(* PLC project Unnamed, Unknown Unnamed 1 *)
(* stored: creationDateTime 2025-11-14T09:55:49, modificationDateTime 2026-02-01T23:59:25 *)

PROGRAM program0
  VAR
    TP0 : TP;  (* Pulse Timer *)
  END_VAR
  VAR
    InletValve1 AT %QX0.1 : BOOL;  (* Output *)
    InletValve2 AT %QX0.2 : BOOL;  (* Output *)
    Start AT %IX0.1 : BOOL;  (* Input *)
    Stop AT %IX0.2 : BOOL;  (* Input *)
    CycleOn AT %IX0.3 : BOOL;  (* Input *)
    LevelSensor1 AT %IX0.4 : BOOL;  (* Input *)
    LevelSensor2 AT %IX0.5 : BOOL;  (* Input *)
    AgitatorMotor AT %QX0.3 : BOOL;  (* Output *)
    LowLevelSensor AT %IX0.6 : BOOL;  (* Input *)
    OutletValve AT %QX0.4 : BOOL;  (* Output *)
    TemperatureSensor AT %IW0 : INT := 28;  (* Input *)
  END_VAR
  VAR
    Flag : BOOL;
  END_VAR
  VAR
    Heater AT %QX1.0 : BOOL;  (* Output *)
  END_VAR

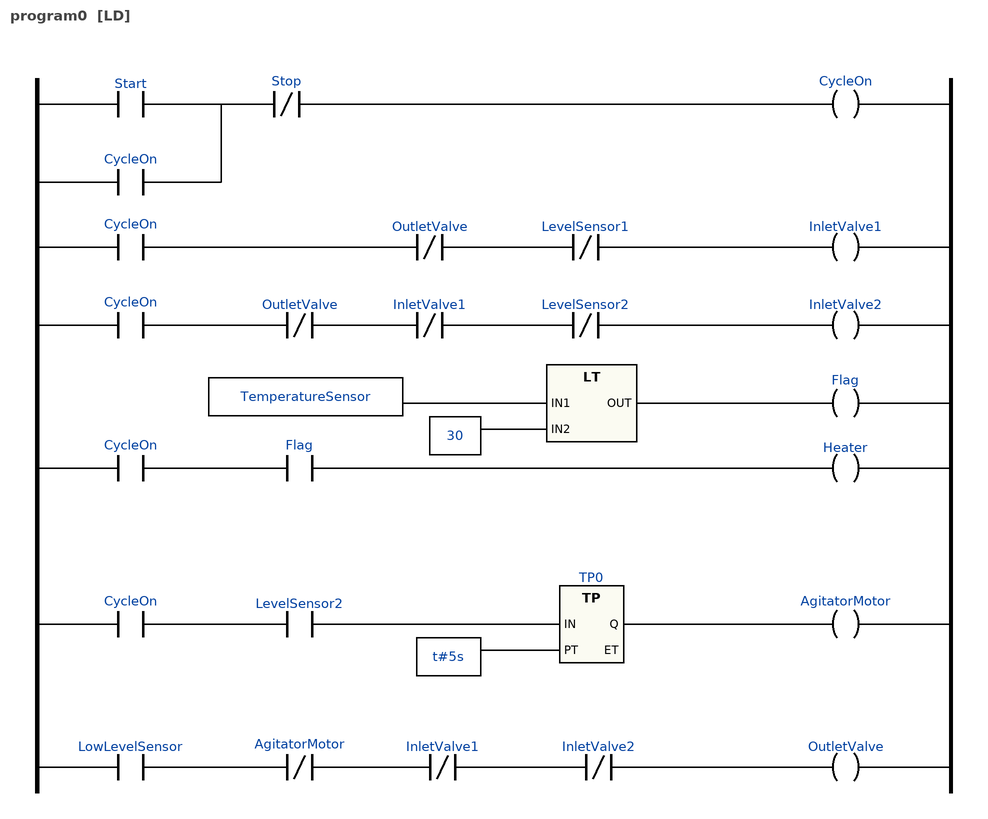
(* LD diagram, written out as Structured Text *)
CycleOn := (Start OR CycleOn) AND NOT Stop;
InletValve1 := CycleOn AND NOT OutletValve AND NOT LevelSensor1;
InletValve2 := CycleOn AND NOT OutletValve AND NOT InletValve1 AND NOT LevelSensor2;
TP0(IN := CycleOn AND LevelSensor2, PT := t#5s);
AgitatorMotor := TP0.Q;
OutletValve := LowLevelSensor AND NOT AgitatorMotor AND NOT InletValve1 AND NOT InletValve2;
Flag := TemperatureSensor < 30;
Heater := CycleOn AND Flag;
END_PROGRAM

CONFIGURATION Config0
  RESOURCE Res0 ON PLC
    TASK task0(INTERVAL := T#20ms, PRIORITY := 0);
    PROGRAM instance0 WITH task0 : program0;
  END_RESOURCE
END_CONFIGURATION
